// SIMATIC S7-200 project (STEP 7-Micro/WIN), CPU 214 REL 01.11

ORGANIZATION_BLOCK MAIN:OB1
TITLE=这个项目包含自动化仓库货架小车运动控制模块。控制设备包括前后电动机、升降机和货叉伸缩机构。 小车配备前后电动机、升降机和货叉伸缩机构。
// 操作员通过手自动按钮选择手动或自动模式，当前模式由手自动切换标志指示。在自动模式下，系统根据预设的目标列计数和目标行计数引导小车移动。首先，小车通过前后电动机向前运动信号移动到指定列，系统持续比较当前列计数与目标列计数，只有两者相等时，才会触发前后电动机向前停止信号并置位前后运动到位标志。随后，升降机启动，只有在前后运动到位标志置位后，升降机上升信号才会激活，系统监控当前行计数与目标行计数，当两者相等时，触发升降机上升停止信号并置位升降运动到位标志。
// 到达目标位置后，小车继续执行货叉动作。只有在前后运动到位标志和升降运动到位标志都置位的情况下，货叉前伸信号才会触发，货叉伸出，动作时间由货叉伸缩定时器控制，例如3.6秒完成30厘米伸缩，到时后置位货叉伸缩到位标志。接下来，根据货叉动作选择的状态，ON表示放下，OFF表示抓取，只有在货叉伸缩到位标志置位后，系统才会激活货叉放下货物信号或货叉抓取货物信号，完成货物的存取。任务完成后，当前后运动到位标志、升降运动到位标志和货叉伸缩到位标志全部置位时，返回标志被置位，小车通过前后电动机向后运动信号和升降机下降信号返回初始位置。
// 在手动模式下，操作员通过一系列按钮直接控制小车。例如，手动向前运动标志和前后电动机运行按钮必须同时为ON，才能触发前后电动机向前运动信号；若前后电动机运行按钮为OFF，则触发前后电动机向前停止信号并置位前后运动到位标志。类似地，手动上升运动标志或手动下降运动标志控制升降机，手动货叉前伸标志或手动货叉后退标志控制货叉，确保操作员能够灵活调整小车位置。
// 
// 
BEGIN
Network 1
// 
//  
// 
LD     SM0.0
CALL   singal:SBR0
?000
Network 2
// M0.0手自动按钮   M0.0的数值是由开关量输入模块读入的
Network 3
// M10.0  手自动切换                         M20.0  前后电动机运行按钮        -----------------以下自动运行 L3----------L4
LD     SM0.0
LPS
AN     M20.7
AN     M20.1
A      M0.0
A      M10.0
S      Q0.0, 0
LPP
A      M20.7
AN     M20.5
AN     M20.3
A      M0.0
A      M10.0
S      Q0.2, 0
Network 4
// 当VD100 == VD120时，也就是当测量到的列数计数与输入设定列数相等时，停止前后运动电机,同时设置M20.1
// 定义M20.1为前后运动到位标志
LD     SM0.0
LPS
AN     M20.7
AN     M20.1
A      M0.0
A      M10.0
AD=    VD102, VD120
=      Q0.1
S      M20.1, 0
LPP
A      M20.7
AN     M20.5
AN     M20.3
A      M0.0
A      M10.0
AD=    VD102, VD120
=      Q0.3
R      M20.1, 0
Network 5
// 以下手动控制小车前后运动 M21.0 读取自开关量输入，为向前运动标志
// 因为手动控制有可能会超过预想的位置，下面是手动向后运行的部分
// M21.1 为向后运动标志
LD     SM0.0
A      M0.0                  //如果处于运行状态 (M0.0 为ON)  
AN     M10.0                 //当M10.0为OFF时，表示处于手动控制状态
LPS
A      M21.0                 //如果M21.0为ON,表示小车进行向前运行动作
LPS
A      M20.0                 //如果此时按下前后运动电机启动按钮
S      Q0.0, 0               //那么将输出向前运动信号，使小车向前运动
LPP
AN     M20.0                 //如果此时前后电机运行按钮时停止的
=      Q0.1                  //那么将输出向前运动停止信号，小车停止前进
S      M20.1, 0              //同时设置M20.1,表明小车前后运动已经完成。
LPP
A      M21.1                 //存在向前的同时就可能存在向后的运动
LPS
A      M20.0                 //如果启动前后运行电机
S      Q0.2, 0               //那么将输出向后运行信号，小车向后运动
LPP
AN     M20.0                 //如果此时前后电机运行按钮是停止的
=      Q0.3                  //那么将输出向后运动停止信号，小车停止后退
S      M20.1, 0              //同时设置M20.1,表明小车前后运动已经完成。
Network 6
// 下面控制上下运动，按原理分析，上下运动的控制与前后运动是相同的  M20.2 为上下运动使能标志
LD     SM0.0
LPS
AN     M20.7                 //如果M20.7为OFF，表明小车在前进完成任务的过程中
A      M20.1                 //如果M20.1为ON,表明小车已经完成了前后方向的运行
AN     M20.3                 //M20.3为OFF,表明机械手还没有完成升降运行的动作
A      M0.0                  //M0.0为ON,表明"START"按钮已经按下，处于运动过程中
A      M10.0                 //M10.0为ON,小车处于自动控制状态
S      Q0.4, 0               //输出信号，机械手臂抬升货物
LPP
A      M20.7                 //如果M20.7为ON，表明小车已经完成了预定动作，返回
AN     M20.5                 //如果M20.5为OFF,表明机械手臂完成了存取货物返回的动作
A      M0.0                  //如果M0.0为ON（START按下）
A      M10.0                 //自动运行状态
S      Q0.6, 0               //那么输出信号，机械手执行下降动作
Network 7
LD     SM0.0
LPS
AN     M20.7                 //前进过程中
A      M20.1
AN     M20.3
A      M0.0
A      M10.0
AR=    VD100, VD150          //当测量到的行计数与输出的设定行数相等时，
//认为已经达到了预定的行数位置，那么停止小车上升运动
=      Q0.5
S      M20.3, 0              //同时设置行位置已经达到标志M20.3
LPP
A      M20.7                 //返回过程中
AN     M20.5
A      M0.0
A      M10.0
AD=    VD100, VD150          //当测量到的行计数与输出的设定行数相等时，
S      Q0.7, 0
R      M20.3, 0              //认为机械手已经降到原始位置，所以清除行位置达到标志
Network 8
LD     SM0.0
A      M0.0                  //如果处于运行状态 (M0.0 为ON) 
AN     M10.0                 //当M10.0为OFF时，表示处于手动控制状态
LPS
A      M21.2                 //如果M21.2为ON,表示小车进行向上升运行
LPS
A      M20.2                 //如果此时允许机械手升降运动
S      Q0.4, 0               //那么将输出向上运动信号，使小车上升运动
LPP
AN     M20.2                 //如果此时升降电机运行按钮时停止的
=      Q0.5
S      M20.3, 0              //那么将输出上升运动停止信号，小车停止上升
LPP
A      M21.3
LPS
A      M20.2                 //如果启动升降运行电机
S      Q0.6, 0               //那么将输出下降运行信号，机械手向下运动
LPP
AN     M20.2                 //如果此时升降电机运行按钮是停止的
=      Q0.7                  //那么将输出向下运动停止信号，小车停止下降
S      M20.3, 0              //同时设置M20.3,表明小车升降运动已经完成。
Network 9
// 以上程序完成小车前后、升降的运动，下面是机械手臂的伸缩运动  --自动控制部分
LD     SM0.0
LPS
AN     M20.7                 //前进过程中
A      M20.1                 //已经到达了指定的列       
A      M20.3                 //已经到达了指定的行
A      M0.0                  //运行状态
A      M10.0                 //自动状态
S      Q1.0, 0               //控制机械手臂前伸
LPP
A      M20.7                 //返回过程中
A      M20.5                 //还没有完成机械手回缩的动作
A      M0.0                  //运行状态
A      M10.0                 //自动状态
S      Q1.2, 0               //输出信号，机械手后退，离开货架
Network 10
// 当伸缩手臂开始向前运动时，假设其36 * 100 MS      3.6S = 0.06MIN  L = 0.06* 5 =  30CM    
LD     SM0.0
LPS
AN     M20.7                 //前进过程中
A      M20.1                 //已经到达指定列
A      M20.3                 //已经到达指定行
A      M0.0                  //开始运行
A      M10.0                 //自动运行状态
AN     M20.5                 //机械手存取动作未完成
TON    T37, +36              //设置100MS定时器。
LPP
A      M20.7                 //返回过程中。
A      M20.5                 //机械手存取动作已经完成
A      M0.0
A      M10.0
TON    T37, +36              //设置100MS定时器。     
Network 11
// 定时器时间到，认为手臂已经到达指定位置
LD     SM0.0
LPS
AN     M20.7                 //如果未完成存取物品动作
A      M20.1                 //已经到达指定列
A      M20.3                 //已经到达指定行
A      M0.0                  //开始运行
A      M10.0                 //自动运行
A      T37                   //如果定时器时间已到
S      M20.5, 0              //认为机械手已经到达货架指定位置,输出信号停止机械手运动
=      Q1.1                  //设置机械手到达货架指定位置标志M20.5
LPP
A      M20.7                 //在返回途中
A      M20.1
A      M20.3
A      M20.5
A      M0.0
A      M10.0
A      T37                   //如果定时器时间到
R      M20.5, 0              //清除机械手到位标志
S      Q1.3, 0               //同时停止机械手运动
Network 12
// 将货物放下Q1.4控制将货物放下 Q1.5抓起货物   M22.0 为抓取或放下的选择条件，ON时放下
LD     SM0.0
AN     M20.7                 //未完成存取物品的动作时
A      M20.5                 //如果机械手已经到达了货架的指定位置
A      M0.0
A      M10.0
LPS
A      M22.0                 //M22.0为ON表示机械手放下货物标志
S      Q1.4, 0               //输出信号，使机械手放下货物
LPP
AN     M22.0                 //M22.0为OFF表示机械手抓取货物标志
S      Q1.5, 0               //输出信号，使机械手抓取货物
Network 13
// 手动部分 伸
LD     SM0.0
A      M0.0
AN     M10.0                 //手动控制
LPS
A      M21.4                 //M21.4为向前运动标志
LPS
A      M20.4                 //如果机械手伸缩按钮按下
S      Q1.0, 0               //那么输出信号使机械手前伸
LPP
AN     M20.4                 //如果机械手伸缩按钮弹起
=      Q1.1                  //那么输出信号使机械手停止前伸
S      M20.5, 0              //设置机械手伸缩运动到位标志
LPP
A      M21.5                 //如果机械手向后运动标志ON
LPS
A      M20.4                 //如果按钮按下
S      Q1.2, 0               //输出信号使机械手后退       
LPP
AN     M20.4                 //如果机械手伸缩按钮弹起
=      Q1.3                  //那么输出信号使机械手停止后退
S      M20.5, 0              //同时清除机械手到位标志
Network 14
// 如果M20.1; M20.3;M20.5 三个标志都被设置成为1，那么认为现在处于放置完或者取完货物状态，下面的程序是
// 返回的部分，M20.7 是 返回标志
LD     SM0.0
A      M20.1
A      M20.3
A      M20.5
S      M20.7, 0              //如果M20.1 M20.3 M20.5都为ON,那么认为
//已经完成了存放物品的整个过程，设置
//运行标志位作为返回程序的标志
END_ORGANIZATION_BLOCK

SUBROUTINE_BLOCK singal:SBR0
TITLE=POU Comment
BEGIN
Network 1 // 初始化
//  
// NETWORK COMMENTS
//  
// 
LD     SM0.1
MOVW   +0, VW102
MOVW   +0, VW132
Network 2 // AIW0为层数
// 
// 
LD     SM0.0
MOVW   AIW0, VW102
Network 3 //   
// 
// 
LDW>=  VW102, +0
MOVW   +0, VW100
NOT
MOVW   16#FFFF, VW100
Network 4 // 累加16次   求和
// 
// 
LD     SM0.0
+D     VD100, VD108
INCB   MB7
Network 5
LDB>=  MB7, 16
MOVD   VD108, VD112
Network 6 // 取平均值
// 
// 
LDB>=  MB7, 16
SRD    VD112, 4
Network 7
LDB>=  MB7, 16
MOVD   +0, VD108
MOVB   0, MB7
Network 8
LD     SM0.0
MOVD   VD112, VD116
Network 9 // 层数VD120
// 
// 
LD     SM0.0
DTR    VD116, VD120
Network 11 // AIW2为列数
// 
// 
LD     SM0.0
MOVW   AIW2, VW132
Network 12 //   
// 
// 
LDW>=  VW132, +0
MOVW   +0, VW130
NOT
MOVW   16#FFFF, VW130
Network 13 // 累加16次   求和
// 
// 
LD     SM0.0
+D     VD130, VD138
INCB   MB10
Network 14
LDB>=  MB10, 16
MOVD   VD138, VD142
Network 15 // 取平均值
// 
// 
LDB>=  MB10, 16
SRD    VD142, 4
Network 16
LDB>=  MB10, 16
MOVD   +0, VD138
MOVB   0, MB10
Network 17
LD     SM0.0
MOVD   VD142, VD146
Network 18 // 层数VD120
// 
// 
LD     SM0.0
DTR    VD146, VD150
Network 19
LD     M20.7
MOVD   +0, VD120
MOVD   +0, VD150
Network 32 // Network Title
// Network Comment
Network 57 // 初始化
//  
// NETWORK COMMENTS
//  
// 
Network 58 // AIW0为烟道温度    AIW2为蒸汽压力    
// 
// 
Network 59 // 烟道温度   
// 
// 
Network 60 // 蒸汽压力  
// 
// 
Network 61 // 累加16次   求和
// 
// 
Network 63 // 取平均值
// 
// 
Network 66 // 烟道温度变送器的量程为0-350℃
// 
// 
Network 67 // 蒸汽压力变送器的量程为0-2.0Mpa
// 
// 
Network 84 // Network Title
// Network Comment
END_SUBROUTINE_BLOCK
